{attribute addProperty BoxType "AT2026-0250-0020"}
{attribute addProperty Id "A_0078_AT2001_5250_0019_AT2001_5250AT2001_3DCFC8D064080"}
{attribute addProperty CRC "1513173855"}
{attribute addProperty SizeInBites "640"}
{attribute addProperty SizeInBytes "80"}
TYPE A_0066_AT2026_0250_0020_AT2026_0250_5A31335F EXTENDS AT2026_9506A482 :
STRUCT
	{attribute addProperty Name "A_0078_AT2001_5250_0019_AT2001_5250"}
	A_0078_AT2001_5250_0019_AT2001_5250 : AT2001_3DCFC8D0;
END_STRUCT
END_TYPE

(* stored: Version 1.2.0.0, ProductVersion 3.1.4024.9
   DUT A_0066_AT2026_0250_0020_AT2026_0250_5A31335F: Id {c9bcf5e2-eba7-462a-8257-eae9bea04e2d} *)
